// TIA Portal V20 export
// export: Created 2026-07-10T11:12:34.52223Z, ExportSetting WithDefaults, DisplayName Totally Integrated Automation Portal, DisplayVersion V20, DisplayName TIA Portal Openness, DisplayVersion V20, DisplayName TIA Portal Version Control Interface, DisplayVersion V20, DisplayName STEP 7 Professional, DisplayVersion V20, DisplayName STEP 7 Safety, DisplayVersion V20, DisplayName WinCC Basic/Comfort/Advanced, DisplayVersion V20, DisplayName WinCC Unified, DisplayVersion V20
FUNCTION_BLOCK "TankWeigher"   // FB25, SCL
{ S7_Optimized_Access := 'TRUE' }
VERSION : 0.1
// stored: AutoNumber true, IsIECCheckEnabled false, IsRetainMemResEnabled false, MemoryReserve 100, SetENOAutomatically false, UDAEnableTagReadback false
   VAR_INPUT
      WeightDelay : Time := T#30s;
      WeightDeadZone : Real := 0.1;
      DayTour : Int;
      CalendarDay : UInt;
      CalendarMonth : UInt;
   END_VAR
   VAR_OUTPUT
      IsWeightMessured : Bool;
      IsFeedLoaded : Bool;
      IsFeedConsumed : Bool;
   END_VAR
   VAR_IN_OUT
      ref_RetainData : "WeightRetainData";
   END_VAR
   VAR
      TankDetector1 { S7_SetPoint := 'True'} : "TankDetector";
      TankRegistrator1 { S7_SetPoint := 'True'} : "TankRegistrator";
      TankDetector2 { S7_SetPoint := 'True'} : "TankDetector";
   END_VAR
BEGIN
   #TankDetector1(WeightValue:="MB".Table.WeightValue1,
                  WeightDelay:=#WeightDelay,
                  WeightError:=false,
                  DeadZone:=#WeightDeadZone,
                  IsWeightMeasured=>#IsWeightMessured,
                  IsFeedLoaded=>#IsFeedLoaded,
                  IsFeedConsumed=>#IsFeedConsumed,
                  Ref_ConsumedFeed:=#ref_RetainData.ConsumedFeed1,
                  Ref_LoadedFeed:=#ref_RetainData.LoadedFeed1,
                  Ref_PreviousWeight:=#ref_RetainData.PreviousWeight1);

   #TankDetector2(WeightValue := "MB".Table.WeightValue2,
                  WeightDelay := #WeightDelay,
                  WeightError := false,
                  DeadZone := #WeightDeadZone,
                  IsWeightMeasured => #IsWeightMessured,
                  IsFeedLoaded => #IsFeedLoaded,
                  IsFeedConsumed => #IsFeedConsumed,
                  Ref_ConsumedFeed := #ref_RetainData.ConsumedFeed2,
                  Ref_LoadedFeed := #ref_RetainData.LoadedFeed2,
                  Ref_PreviousWeight := #ref_RetainData.PreviousWeight2);

   #TankRegistrator1(CurrentConsumedFeed1:=#ref_RetainData.ConsumedFeed1,
                     CurrentConsumedFeed2:=#ref_RetainData.ConsumedFeed2,
                     CurrentLoadedFeed1:=#ref_RetainData.LoadedFeed1,
                     CurrentLoadedFeed2:=#ref_RetainData.LoadedFeed2,
                     DayTour:=#DayTour,
                     CalendarDay:=#CalendarDay,
                     CalendarMonth:=#CalendarMonth,
                     ref_RetainData:=#ref_RetainData);


   IF #TankRegistrator1.ResetCounters THEN
       #TankDetector1.Ref_ConsumedFeed := 0;
       #TankDetector1.Ref_LoadedFeed := 0;
       #TankDetector1.Ref_PreviousWeight := 0;
       #TankDetector2.Ref_ConsumedFeed := 0;
       #TankDetector2.Ref_LoadedFeed := 0;
       #TankDetector2.Ref_PreviousWeight := 0;
   END_IF;
END_FUNCTION_BLOCK
